// Implicitly generated code : DO NOT EDIT
FUNCTION CheckDivLInt : LINT
VAR_INPUT
	divisor:LINT;
END_VAR

// Implicitly generated code : Only an Implementation suggestion
{noflow}
IF divisor = 0 THEN
GVL_Checks.diCheckDivLInt := GVL_Checks.diCheckDivLInt +1;
	CheckDivLInt:=1;
ELSE
	CheckDivLInt:=divisor;
END_IF;
{flow}

END_FUNCTION

(* stored: Version 1.1.0.1, ProductVersion 3.1.4024.12
   POU CheckDivLInt: Id {a77c8f14-2e66-42d1-8fb9-9e0442b706cd}, SpecialFunc CheckDivInt64 *)
